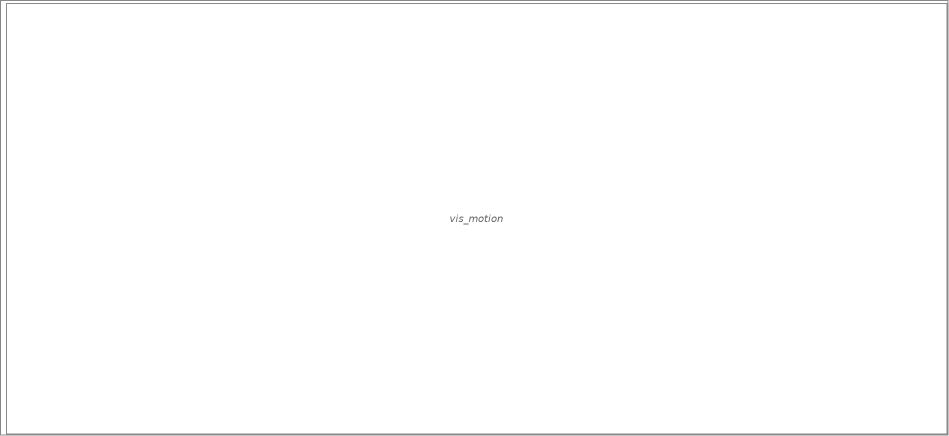
VISUALIZATION main_tabs  // 949x436
    TabControl (6,3 941x431)
        shows vis_motion()
        shows vis_calibration()
        [0]: TabTitle=Motion
        [1]: TabTitle=Calibration
END_VISUALIZATION

(* stored: Version 1.1.0.1, ProductVersion 3.1.4024.0
   Visu main_tabs: Id {04b9e198-3a60-4e84-9ad1-495d6d1eb211} *)
